(*
A tool for performing CASE OF-like evaluations on `I_Tag`.  
It enables sequential evaluation of conditions and stops when `IsTrue`, `IsFalse`, or `IsErr` methods are invoked.
Allows method chaining.
*)
INTERFACE INTERNAL I_TagCmp

(*
Updates its internal state based on the internal status and option.  
Sets the state to `Ok` if the base tag is `Ok` and has the specified Option; otherwise, sets the state to `None`.
*)
METHOD AndHasOption : I_TagCmp
VAR_INPUT
	sOption		: Str;
END_VAR
END_METHOD

(*
Updates its internal state based on the internal status and an external condition.  
Sets the state to `Ok` if the base tag is `Ok` and the external condition is TRUE; otherwise, sets the state to `None`.
*)
METHOD AndIf : I_TagCmp
VAR_INPUT
	bCondition: BOOL;
END_VAR
END_METHOD

(*
Updates its internal state based on the internal status and option.  
Sets the state to `Ok` if the base tag has the specified Option.
*)
METHOD HasOption : I_TagCmp
VAR_INPUT
	sOption		: Str;
END_VAR
END_METHOD

(*
Returns `TRUE` if any evaluated conditions resulted in `Error`.  
Halts further evaluations by locking the current state.
*)
METHOD IsErr : BOOL
VAR_INPUT
END_VAR
END_METHOD

(*
Returns `TRUE` if all evaluated conditions resulted in `FALSE`.  
Halts further evaluations by locking the current state.
*)
METHOD IsFalse : BOOL
VAR_INPUT
END_VAR
END_METHOD

(*
Returns `TRUE` if any evaluated condition resulted in `TRUE`.  
Halts further evaluations by locking the current state.
*)
METHOD IsTrue : BOOL
VAR_INPUT
END_VAR
END_METHOD

(*
Updates its internal state based on the internal status and external I_Tag.  
Sets the state to `Ok` if the base tag matches the external tag.
*)
METHOD Match : I_TagCmp
VAR_INPUT
	iOther: I_Tag;
END_VAR
END_METHOD

(*
Updates its internal state based on the internal status and a string value.  
Sets the state to `Ok` if the base tag Id matches the provided string from right to left.
*)
METHOD MatchId : I_TagCmp
VAR_INPUT
	sIdToMatch		: Str;
END_VAR
END_METHOD

(*
Updates its internal state based on the internal status and a string value.  
Sets the state to `Ok` if the base tag Id matches the provided string pattern.
Allows wildcards.
*)
METHOD MatchWcdId : I_TagCmp
VAR_INPUT
	sPattern 			: Str;
END_VAR
END_METHOD

(*
Updates its internal state based on the internal status and an external condition.  
Sets the state to `Ok` if the base tag is `Ok` or the external condition is TRUE.
*)
METHOD OrIf : I_TagCmp
VAR_INPUT
	bCondition: BOOL;
END_VAR
END_METHOD

(*
Sets a new base tag for comparison and resets the result and lock states.
Fails if `iBaseTag` is `0`;
*)
METHOD Set : I_TagCmp
VAR_INPUT
	iBaseTag	: I_Tag;
END_VAR
END_METHOD

(*
Updates its internal state based on the internal status and an external condition.  
Sets the state to `Ok` if the base tag is `Ok` xor the external condition is TRUE.
*)
METHOD XorIf : I_TagCmp
VAR_INPUT
	bCondition: BOOL;
END_VAR
END_METHOD

END_INTERFACE

(* stored: Version 1.1.0.1
   Itf I_TagCmp: Id {434164ab-6703-48fd-8c7c-cbf390d14597}
   Method AndHasOption: Id {a4585c99-f8a4-4b83-ba90-93fe3a2200bf}
   Method AndIf: Id {436de305-153d-45a1-9c24-e403a9752ee1}
   Method HasOption: Id {b84f95c7-a356-49dc-93c9-34f52a63a0d6}
   Method IsErr: Id {eade2c83-2eb4-4906-a88c-ecc02bd7617e}
   Method IsFalse: Id {1ddd5fe7-59a2-41d0-a2b4-4e9b08b22807}
   Method IsTrue: Id {34600bc9-ed75-446f-8d26-ff01d90d3395}
   Method Match: Id {ff272183-aeae-424d-9c25-2144ef81905e}
   Method MatchId: Id {5cba49aa-7253-4bc9-829c-d83e4b3c65d2}
   Method MatchWcdId: Id {babfa847-1376-48d8-8950-170aa75af813}
   Method OrIf: Id {43b0b3b9-ad9a-4aeb-88cb-22e31aac3fe8}
   Method Set: Id {94ae1389-8107-4a7f-b005-7ced5ba44f46}
   Method XorIf: Id {d8e35498-785d-4895-9e65-30990ff7fe09} *)
